// TIA Portal V18 export
TYPE "UDT_OP10_Recipe_diff"
   STRUCT
      Header : Struct   // Information about recipe
         RecipeName : Bool;
         RecipeID : Bool;
         "Version" : Bool;
         LastModified : Bool;
         PartType : Bool;
         PartTypeRecordNr : Bool;
      END_STRUCT;
      Process : Struct   // Important process parameters how should machine act
         Timers : Struct   // Definition of times for processess
            Delay_Short : Bool;
            Delay_Medium : Bool;
            Delay_Long : Bool;
            Cylinder_ActTime : Bool;
         END_STRUCT;
         Limits : Struct   // limitations of the values
            RetryLimit : Bool;
         END_STRUCT;
         Press : Struct   // parameters for the kistler press devices
            B1_Program : Bool;
            B2_Program : Bool;
            Curve : Struct
               StartPos_UL : Bool;
               StartPos_LL : Bool;
               StartForce_UL : Bool;
               StartForce_LL : Bool;
               MiddlePos_UL : Bool;
               MiddlePos_LL : Bool;
               MiddleForce_UL : Bool;
               MiddleForce_LL : Bool;
               FinalPos_UL : Bool;
               FinalPos_LL : Bool;
               FinalForce_UL : Bool;
               FinalForce_LL : Bool;
               ProgramNum : Bool;
            END_STRUCT;
         END_STRUCT;
         Vision : Struct   // camera system programs numbers
            CGlueShaftIV3_Progs : Array[1..4] of Bool;
            CGlueMagnetIV3_Prog : Bool;
            CGlueProgram : Bool;
         END_STRUCT;
      END_STRUCT;
      "Tooling Code" : Struct   // QR CODES OF THE TOOLING FOR THE RECIPE
         A1_Table : Array[0..10] of Bool;
         A2_Table : Array[0..10] of Bool;
         ROB1_Shaft_Handling_Robot : Struct   // R1
            Gripper : Struct
               "JAW TOOLING LEFT" : Bool;
               "JAW TOOLING RIGHT" : Bool;
               "SHAFT CLAMPING LEFT" : Bool;
               "SHAFT CLAMPING RIGHT" : Bool;
            END_STRUCT;
         END_STRUCT;
         ROB2_Main_Assembly_Robot : Struct   // R2
            Gripper : Struct
               "JAW TOOLING LEFT" : Bool;
               "JAW TOOLING RIGHT" : Bool;
               "SHAFT CLAMPING LEFT" : Bool;
               "SHAFT CLAMPING RIGHT" : Bool;
            END_STRUCT;
         END_STRUCT;
         ROB3_Unloading_Robot : Struct   // R3
            Gripper : Struct
               "JAW TOOLING LEFT" : Bool;
               "JAW TOOLING RIGHT" : Bool;
               "SHAFT CLAMPING LEFT" : Bool;
               "SHAFT CLAMPING RIGHT" : Bool;
            END_STRUCT;
         END_STRUCT;
      END_STRUCT;
      Motion : Struct   // ALL SERVO DRIVES PARAMETERS
         Gluing_Nozzle_Z : Struct   // Physical Axis: IAI_A1
            Position_01 : Struct
               Pos : Bool;
               Vel : Bool;
            END_STRUCT;
            Position_02 : Struct
               Pos : Bool;
               Vel : Bool;
            END_STRUCT;
            Position_03 : Struct
               Pos : Bool;
               Vel : Bool;
            END_STRUCT;
            Position_04 : Struct
               Pos : Bool;
               Vel : Bool;
            END_STRUCT;
            Position_05 : Struct
               Pos : Bool;
               Vel : Bool;
            END_STRUCT;
            Position_06 : Struct
               Pos : Bool;
               Vel : Bool;
            END_STRUCT;
            Position_07 : Struct
               Pos : Bool;
               Vel : Bool;
            END_STRUCT;
            Position_08 : Struct
               Pos : Bool;
               Vel : Bool;
            END_STRUCT;
            Position_09 : Struct
               Pos : Bool;
               Vel : Bool;
            END_STRUCT;
            Position_10 : Struct
               Pos : Bool;
               Vel : Bool;
            END_STRUCT;
            Position_11 : Struct
               Pos : Bool;
               Vel : Bool;
            END_STRUCT;
            Position_12 : Struct
               Pos : Bool;
               Vel : Bool;
            END_STRUCT;
            Position_13 : Struct
               Pos : Bool;
               Vel : Bool;
            END_STRUCT;
            Position_14 : Struct
               Pos : Bool;
               Vel : Bool;
            END_STRUCT;
            Position_15 : Struct
               Pos : Bool;
               Vel : Bool;
            END_STRUCT;
            Position_16 : Struct
               Pos : Bool;
               Vel : Bool;
            END_STRUCT;
            Position_17 : Struct
               Pos : Bool;
               Vel : Bool;
            END_STRUCT;
            Position_18 : Struct
               Pos : Bool;
               Vel : Bool;
            END_STRUCT;
            Position_19 : Struct
               Pos : Bool;
               Vel : Bool;
            END_STRUCT;
            Position_20 : Struct
               Pos : Bool;
               Vel : Bool;
            END_STRUCT;
         END_STRUCT;
         Gluing_Nozzle_X : Struct   // Physical Axis: IAI_A2
            Position_01 : Struct
               Pos : Bool;
               Vel : Bool;
            END_STRUCT;
            Position_02 : Struct
               Pos : Bool;
               Vel : Bool;
            END_STRUCT;
            Position_03 : Struct
               Pos : Bool;
               Vel : Bool;
            END_STRUCT;
            Position_04 : Struct
               Pos : Bool;
               Vel : Bool;
            END_STRUCT;
            Position_05 : Struct
               Pos : Bool;
               Vel : Bool;
            END_STRUCT;
            Position_06 : Struct
               Pos : Bool;
               Vel : Bool;
            END_STRUCT;
            Position_07 : Struct
               Pos : Bool;
               Vel : Bool;
            END_STRUCT;
            Position_08 : Struct
               Pos : Bool;
               Vel : Bool;
            END_STRUCT;
            Position_09 : Struct
               Pos : Bool;
               Vel : Bool;
            END_STRUCT;
            Position_10 : Struct
               Pos : Bool;
               Vel : Bool;
            END_STRUCT;
            Position_11 : Struct
               Pos : Bool;
               Vel : Bool;
            END_STRUCT;
            Position_12 : Struct
               Pos : Bool;
               Vel : Bool;
            END_STRUCT;
            Position_13 : Struct
               Pos : Bool;
               Vel : Bool;
            END_STRUCT;
            Position_14 : Struct
               Pos : Bool;
               Vel : Bool;
            END_STRUCT;
            Position_15 : Struct
               Pos : Bool;
               Vel : Bool;
            END_STRUCT;
            Position_16 : Struct
               Pos : Bool;
               Vel : Bool;
            END_STRUCT;
            Position_17 : Struct
               Pos : Bool;
               Vel : Bool;
            END_STRUCT;
            Position_18 : Struct
               Pos : Bool;
               Vel : Bool;
            END_STRUCT;
            Position_19 : Struct
               Pos : Bool;
               Vel : Bool;
            END_STRUCT;
            Position_20 : Struct
               Pos : Bool;
               Vel : Bool;
            END_STRUCT;
         END_STRUCT;
         Gluing_Nozzle_Y : Struct   // Physical Axis: IAI_A3
            Position_01 : Struct
               Pos : Bool;
               Vel : Bool;
            END_STRUCT;
            Position_02 : Struct
               Pos : Bool;
               Vel : Bool;
            END_STRUCT;
            Position_03 : Struct
               Pos : Bool;
               Vel : Bool;
            END_STRUCT;
            Position_04 : Struct
               Pos : Bool;
               Vel : Bool;
            END_STRUCT;
            Position_05 : Struct
               Pos : Bool;
               Vel : Bool;
            END_STRUCT;
            Position_06 : Struct
               Pos : Bool;
               Vel : Bool;
            END_STRUCT;
            Position_07 : Struct
               Pos : Bool;
               Vel : Bool;
            END_STRUCT;
            Position_08 : Struct
               Pos : Bool;
               Vel : Bool;
            END_STRUCT;
            Position_09 : Struct
               Pos : Bool;
               Vel : Bool;
            END_STRUCT;
            Position_10 : Struct
               Pos : Bool;
               Vel : Bool;
            END_STRUCT;
            Position_11 : Struct
               Pos : Bool;
               Vel : Bool;
            END_STRUCT;
            Position_12 : Struct
               Pos : Bool;
               Vel : Bool;
            END_STRUCT;
            Position_13 : Struct
               Pos : Bool;
               Vel : Bool;
            END_STRUCT;
            Position_14 : Struct
               Pos : Bool;
               Vel : Bool;
            END_STRUCT;
            Position_15 : Struct
               Pos : Bool;
               Vel : Bool;
            END_STRUCT;
            Position_16 : Struct
               Pos : Bool;
               Vel : Bool;
            END_STRUCT;
            Position_17 : Struct
               Pos : Bool;
               Vel : Bool;
            END_STRUCT;
            Position_18 : Struct
               Pos : Bool;
               Vel : Bool;
            END_STRUCT;
            Position_19 : Struct
               Pos : Bool;
               Vel : Bool;
            END_STRUCT;
            Position_20 : Struct
               Pos : Bool;
               Vel : Bool;
            END_STRUCT;
         END_STRUCT;
         Ring_Turntable_Axis_1 : Struct   // Physical Axis: V90_A1
            Position_01 : Struct
               Pos : Bool;
               Vel : Bool;
            END_STRUCT;
            Position_02 : Struct
               Pos : Bool;
               Vel : Bool;
            END_STRUCT;
            Position_03 : Struct
               Pos : Bool;
               Vel : Bool;
            END_STRUCT;
            Position_04 : Struct
               Pos : Bool;
               Vel : Bool;
            END_STRUCT;
            Position_05 : Struct
               Pos : Bool;
               Vel : Bool;
            END_STRUCT;
            Position_06 : Struct
               Pos : Bool;
               Vel : Bool;
            END_STRUCT;
            Position_07 : Struct
               Pos : Bool;
               Vel : Bool;
            END_STRUCT;
            Position_08 : Struct
               Pos : Bool;
               Vel : Bool;
            END_STRUCT;
            Position_09 : Struct
               Pos : Bool;
               Vel : Bool;
            END_STRUCT;
            Position_10 : Struct
               Pos : Bool;
               Vel : Bool;
            END_STRUCT;
            Position_11 : Struct
               Pos : Bool;
               Vel : Bool;
            END_STRUCT;
            Position_12 : Struct
               Pos : Bool;
               Vel : Bool;
            END_STRUCT;
            Position_13 : Struct
               Pos : Bool;
               Vel : Bool;
            END_STRUCT;
            Position_14 : Struct
               Pos : Bool;
               Vel : Bool;
            END_STRUCT;
            Position_15 : Struct
               Pos : Bool;
               Vel : Bool;
            END_STRUCT;
            Position_16 : Struct
               Pos : Bool;
               Vel : Bool;
            END_STRUCT;
            Position_17 : Struct
               Pos : Bool;
               Vel : Bool;
            END_STRUCT;
            Position_18 : Struct
               Pos : Bool;
               Vel : Bool;
            END_STRUCT;
            Position_19 : Struct
               Pos : Bool;
               Vel : Bool;
            END_STRUCT;
            Position_20 : Struct
               Pos : Bool;
               Vel : Bool;
            END_STRUCT;
         END_STRUCT;
         Shaft_Scan_Turntable_Axis : Struct   // Physical Axis: V90_A2
            Position_01 : Struct
               Pos : Bool;
               Vel : Bool;
            END_STRUCT;
            Position_02 : Struct
               Pos : Bool;
               Vel : Bool;
            END_STRUCT;
            Position_03 : Struct
               Pos : Bool;
               Vel : Bool;
            END_STRUCT;
            Position_04 : Struct
               Pos : Bool;
               Vel : Bool;
            END_STRUCT;
            Position_05 : Struct
               Pos : Bool;
               Vel : Bool;
            END_STRUCT;
            Position_06 : Struct
               Pos : Bool;
               Vel : Bool;
            END_STRUCT;
            Position_07 : Struct
               Pos : Bool;
               Vel : Bool;
            END_STRUCT;
            Position_08 : Struct
               Pos : Bool;
               Vel : Bool;
            END_STRUCT;
            Position_09 : Struct
               Pos : Bool;
               Vel : Bool;
            END_STRUCT;
            Position_10 : Struct
               Pos : Bool;
               Vel : Bool;
            END_STRUCT;
            Position_11 : Struct
               Pos : Bool;
               Vel : Bool;
            END_STRUCT;
            Position_12 : Struct
               Pos : Bool;
               Vel : Bool;
            END_STRUCT;
            Position_13 : Struct
               Pos : Bool;
               Vel : Bool;
            END_STRUCT;
            Position_14 : Struct
               Pos : Bool;
               Vel : Bool;
            END_STRUCT;
            Position_15 : Struct
               Pos : Bool;
               Vel : Bool;
            END_STRUCT;
            Position_16 : Struct
               Pos : Bool;
               Vel : Bool;
            END_STRUCT;
            Position_17 : Struct
               Pos : Bool;
               Vel : Bool;
            END_STRUCT;
            Position_18 : Struct
               Pos : Bool;
               Vel : Bool;
            END_STRUCT;
            Position_19 : Struct
               Pos : Bool;
               Vel : Bool;
            END_STRUCT;
            Position_20 : Struct
               Pos : Bool;
               Vel : Bool;
            END_STRUCT;
         END_STRUCT;
         Gluing_Rotary_Jig_Axis : Struct   // Physical Axis: V90_A3
            Position_01 : Struct
               Pos : Bool;
               Vel : Bool;
            END_STRUCT;
            Position_02 : Struct
               Pos : Bool;
               Vel : Bool;
            END_STRUCT;
            Position_03 : Struct
               Pos : Bool;
               Vel : Bool;
            END_STRUCT;
            Position_04 : Struct
               Pos : Bool;
               Vel : Bool;
            END_STRUCT;
            Position_05 : Struct
               Pos : Bool;
               Vel : Bool;
            END_STRUCT;
            Position_06 : Struct
               Pos : Bool;
               Vel : Bool;
            END_STRUCT;
            Position_07 : Struct
               Pos : Bool;
               Vel : Bool;
            END_STRUCT;
            Position_08 : Struct
               Pos : Bool;
               Vel : Bool;
            END_STRUCT;
            Position_09 : Struct
               Pos : Bool;
               Vel : Bool;
            END_STRUCT;
            Position_10 : Struct
               Pos : Bool;
               Vel : Bool;
            END_STRUCT;
            Position_11 : Struct
               Pos : Bool;
               Vel : Bool;
            END_STRUCT;
            Position_12 : Struct
               Pos : Bool;
               Vel : Bool;
            END_STRUCT;
            Position_13 : Struct
               Pos : Bool;
               Vel : Bool;
            END_STRUCT;
            Position_14 : Struct
               Pos : Bool;
               Vel : Bool;
            END_STRUCT;
            Position_15 : Struct
               Pos : Bool;
               Vel : Bool;
            END_STRUCT;
            Position_16 : Struct
               Pos : Bool;
               Vel : Bool;
            END_STRUCT;
            Position_17 : Struct
               Pos : Bool;
               Vel : Bool;
            END_STRUCT;
            Position_18 : Struct
               Pos : Bool;
               Vel : Bool;
            END_STRUCT;
            Position_19 : Struct
               Pos : Bool;
               Vel : Bool;
            END_STRUCT;
            Position_20 : Struct
               Pos : Bool;
               Vel : Bool;
            END_STRUCT;
         END_STRUCT;
         Ring_Turntable_Axis_2 : Struct   // Physical Axis: V90_A4
            Position_01 : Struct
               Pos : Bool;
               Vel : Bool;
            END_STRUCT;
            Position_02 : Struct
               Pos : Bool;
               Vel : Bool;
            END_STRUCT;
            Position_03 : Struct
               Pos : Bool;
               Vel : Bool;
            END_STRUCT;
            Position_04 : Struct
               Pos : Bool;
               Vel : Bool;
            END_STRUCT;
            Position_05 : Struct
               Pos : Bool;
               Vel : Bool;
            END_STRUCT;
            Position_06 : Struct
               Pos : Bool;
               Vel : Bool;
            END_STRUCT;
            Position_07 : Struct
               Pos : Bool;
               Vel : Bool;
            END_STRUCT;
            Position_08 : Struct
               Pos : Bool;
               Vel : Bool;
            END_STRUCT;
            Position_09 : Struct
               Pos : Bool;
               Vel : Bool;
            END_STRUCT;
            Position_10 : Struct
               Pos : Bool;
               Vel : Bool;
            END_STRUCT;
            Position_11 : Struct
               Pos : Bool;
               Vel : Bool;
            END_STRUCT;
            Position_12 : Struct
               Pos : Bool;
               Vel : Bool;
            END_STRUCT;
            Position_13 : Struct
               Pos : Bool;
               Vel : Bool;
            END_STRUCT;
            Position_14 : Struct
               Pos : Bool;
               Vel : Bool;
            END_STRUCT;
            Position_15 : Struct
               Pos : Bool;
               Vel : Bool;
            END_STRUCT;
            Position_16 : Struct
               Pos : Bool;
               Vel : Bool;
            END_STRUCT;
            Position_17 : Struct
               Pos : Bool;
               Vel : Bool;
            END_STRUCT;
            Position_18 : Struct
               Pos : Bool;
               Vel : Bool;
            END_STRUCT;
            Position_19 : Struct
               Pos : Bool;
               Vel : Bool;
            END_STRUCT;
            Position_20 : Struct
               Pos : Bool;
               Vel : Bool;
            END_STRUCT;
         END_STRUCT;
      END_STRUCT;
   END_STRUCT;
END_TYPE
